{attribute 'enable_dynamic_creation'}	
{attribute 'no_explicit_call' := 'do not call this function block directly'} 
FUNCTION_BLOCK FileGetCurrentPositionTask EXTENDS FileContentTask
VAR
	_ClassName : STRING := __POUNAME();

    _GetCurrentPosition : Tc2_System.FB_FileTell;
END_VAR

{attribute 'monitoring' := 'call'}
PROPERTY ClassName : STRING
GET
ClassName := _ClassName;
END_GET
END_PROPERTY

METHOD Execute : BOOL
VAR_INPUT
	start : BOOL;
END_VAR
IF start THEN
	Validate();

	_GetCurrentPosition(
		bExecute := FALSE,
		hFile := FilecontentManager.FileHandle,
		sNetId := FilecontentManager.AmsNetId,
		tTimeout := Timeout
	);	
END_IF

_GetCurrentPosition(bExecute := TRUE);

IF _GetCurrentPosition.bError THEN
	//exceptionFactory.ThrowException(__POSITION(), WStringHelper.Concat2("Get current file position failed", GetErrorMessageByErrorId(_GetCurrentPosition.nErrId)), __POUNAME(), ClassName, CurrentNamespace.Name, __POSITION(), _GetCurrentPosition.nErrId);
ELSIF NOT _GetCurrentPosition.bBusy THEN
	Execute := EXECUTION_STATE.DONE;
END_IF
END_METHOD

PROPERTY FilePointerPosition : DINT
GET
FilePointerPosition := _GetCurrentPosition.nSeekPos;
END_GET
END_PROPERTY

END_FUNCTION_BLOCK

(* stored: Version 1.1.0.1
   POU FileGetCurrentPositionTask: Id {cd0a5675-95a4-4646-bcfc-20d965f135d6}, SpecialFunc None
   Property ClassName: Id {ac25b33f-c4ba-4fa3-ae93-4947647d67fd}
   Get Get: Id {88e40f69-2733-46ee-af45-984caca1b3e1}
   Method Execute: Id {8110770f-839c-4bdf-a5d3-5f1503119c05}
   Property FilePointerPosition: Id {db5fd2bf-1abb-4cfa-a475-e1afb32497a7}
   Get Get: Id {fb6630f7-1067-4b15-b49b-0b37e7470dca} *)
